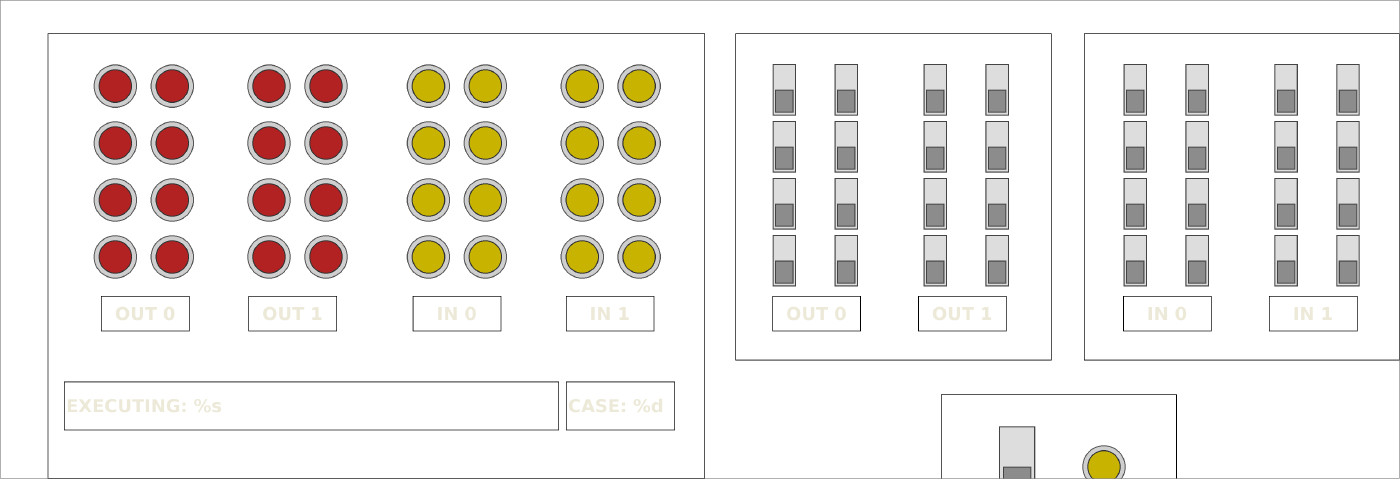
VISUALIZATION StandardPLCversenyVISU  // 1967x673
    Rectangle (1322,554 331x259)
    Rectangle (1033,47 444x459)
    Rectangle (67,47 923x626)
    Lamp1 (127,86 70x70), variable: GIOL.out0, style: Lamp-Lamp1-Red
    Lamp1 (207,86 70x70), variable: GIOL.out1, style: Lamp-Lamp1-Red
    Lamp1 (343,86 70x70), variable: GIOL.out8, style: Lamp-Lamp1-Red
    Lamp1 (423,86 70x70), variable: GIOL.out9, style: Lamp-Lamp1-Red
    Lamp1 (127,166 70x70), variable: GIOL.out2, style: Lamp-Lamp1-Red
    Lamp1 (207,166 70x70), variable: GIOL.out3, style: Lamp-Lamp1-Red
    Lamp1 (343,166 70x70), variable: GIOL.out10, style: Lamp-Lamp1-Red
    Lamp1 (423,166 70x70), variable: GIOL.out11, style: Lamp-Lamp1-Red
    Lamp1 (127,246 70x70), variable: GIOL.out4, style: Lamp-Lamp1-Red
    Lamp1 (207,246 70x70), variable: GIOL.out5, style: Lamp-Lamp1-Red
    Lamp1 (343,246 70x70), variable: GIOL.out12, style: Lamp-Lamp1-Red
    Lamp1 (423,246 70x70), variable: GIOL.out13, style: Lamp-Lamp1-Red
    Lamp1 (127,326 70x70), variable: GIOL.out6, style: Lamp-Lamp1-Red
    Lamp1 (207,326 70x70), variable: GIOL.out7, style: Lamp-Lamp1-Red
    Lamp1 (343,326 70x70), variable: GIOL.out14, style: Lamp-Lamp1-Red
    Lamp1 (423,326 70x70), variable: GIOL.out15, style: Lamp-Lamp1-Red
    Lamp1 (567,86 70x70), variable: GIOL.in0, style: Lamp-Lamp1-Yellow
    Lamp1 (647,86 70x70), variable: GIOL.in1, style: Lamp-Lamp1-Yellow
    Lamp1 (783,86 70x70), variable: GIOL.in8, style: Lamp-Lamp1-Yellow
    Lamp1 (863,86 70x70), variable: GIOL.in9, style: Lamp-Lamp1-Yellow
    Lamp1 (567,166 70x70), variable: GIOL.in2, style: Lamp-Lamp1-Yellow
    Lamp1 (647,166 70x70), variable: GIOL.in3, style: Lamp-Lamp1-Yellow
    Lamp1 (783,166 70x70), variable: GIOL.in10, style: Lamp-Lamp1-Yellow
    Lamp1 (863,166 70x70), variable: GIOL.in11, style: Lamp-Lamp1-Yellow
    Lamp1 (567,246 70x70), variable: GIOL.in4, style: Lamp-Lamp1-Yellow
    Lamp1 (647,246 70x70), variable: GIOL.in5, style: Lamp-Lamp1-Yellow
    Lamp1 (783,246 70x70), variable: GIOL.in12, style: Lamp-Lamp1-Yellow
    Lamp1 (863,246 70x70), variable: GIOL.in13, style: Lamp-Lamp1-Yellow
    Lamp1 (567,326 70x70), variable: GIOL.in6, style: Lamp-Lamp1-Yellow
    Lamp1 (647,326 70x70), variable: GIOL.in7, style: Lamp-Lamp1-Yellow
    Lamp1 (783,326 70x70), variable: GIOL.in14, style: Lamp-Lamp1-Yellow
    Lamp1 (863,326 70x70), variable: GIOL.in15, style: Lamp-Lamp1-Yellow
    Rectangle (349,416 124x49), "OUT 1"
    Rectangle (580,416 124x49), "IN 0"
    Rectangle (142,416 124x49), "OUT 0"
    Rectangle (795,416 124x49), "IN 1"
    Rectangle (90,536 695x68), "EXECUTING: %s", text variable: GIOL.TaskName
    DipSwitch (1153,86 72x80), variable: GIOL.out1, behaviour: TOGGLE, style: Switch-DipSwitch-Gray
    DipSwitch (1066,86 72x80), variable: GIOL.out0, behaviour: TOGGLE, style: Switch-DipSwitch-Gray
    DipSwitch (1153,166 72x80), variable: GIOL.out3, behaviour: TOGGLE, style: Switch-DipSwitch-Gray
    DipSwitch (1066,166 72x80), variable: GIOL.out2, behaviour: TOGGLE, style: Switch-DipSwitch-Gray
    DipSwitch (1153,246 72x80), variable: GIOL.out5, behaviour: TOGGLE, style: Switch-DipSwitch-Gray
    DipSwitch (1066,246 72x80), variable: GIOL.out4, behaviour: TOGGLE, style: Switch-DipSwitch-Gray
    DipSwitch (1153,326 72x80), variable: GIOL.out7, behaviour: TOGGLE, style: Switch-DipSwitch-Gray
    DipSwitch (1066,326 72x80), variable: GIOL.out6, behaviour: TOGGLE, style: Switch-DipSwitch-Gray
    DipSwitch (1365,86 72x80), variable: GIOL.out9, behaviour: TOGGLE, style: Switch-DipSwitch-Gray
    DipSwitch (1278,86 72x80), variable: GIOL.out8, behaviour: TOGGLE, style: Switch-DipSwitch-Gray
    DipSwitch (1365,166 72x80), variable: GIOL.out11, behaviour: TOGGLE, style: Switch-DipSwitch-Gray
    DipSwitch (1278,166 72x80), variable: GIOL.out10, behaviour: TOGGLE, style: Switch-DipSwitch-Gray
    DipSwitch (1365,246 72x80), variable: GIOL.out13, behaviour: TOGGLE, style: Switch-DipSwitch-Gray
    DipSwitch (1278,246 72x80), variable: GIOL.out12, behaviour: TOGGLE, style: Switch-DipSwitch-Gray
    DipSwitch (1365,326 72x80), variable: GIOL.out15, behaviour: TOGGLE, style: Switch-DipSwitch-Gray
    DipSwitch (1278,326 72x80), variable: GIOL.out14, behaviour: TOGGLE, style: Switch-DipSwitch-Gray
    Rectangle (1290,416 124x49), "OUT 1"
    Rectangle (1085,416 124x49), "OUT 0"
    Rectangle (1523,47 444x459)
    DipSwitch (1646,86 72x80), variable: GIOL.bIn1, behaviour: TOGGLE, style: Switch-DipSwitch-Gray
    DipSwitch (1559,86 72x80), variable: GIOL.bIn0, behaviour: TOGGLE, style: Switch-DipSwitch-Gray
    DipSwitch (1646,166 72x80), variable: GIOL.bIn3, behaviour: TOGGLE, style: Switch-DipSwitch-Gray
    DipSwitch (1559,166 72x80), variable: GIOL.bIn2, behaviour: TOGGLE, style: Switch-DipSwitch-Gray
    DipSwitch (1646,246 72x80), variable: GIOL.bIn5, behaviour: TOGGLE, style: Switch-DipSwitch-Gray
    DipSwitch (1559,246 72x80), variable: GIOL.bIn4, behaviour: TOGGLE, style: Switch-DipSwitch-Gray
    DipSwitch (1646,326 72x80), variable: GIOL.bIn7, behaviour: TOGGLE, style: Switch-DipSwitch-Gray
    DipSwitch (1559,326 72x80), variable: GIOL.bIn6, behaviour: TOGGLE, style: Switch-DipSwitch-Gray
    DipSwitch (1858,86 72x80), variable: GIOL.bIn9, behaviour: TOGGLE, style: Switch-DipSwitch-Gray
    DipSwitch (1771,86 72x80), variable: GIOL.bIn8, behaviour: TOGGLE, style: Switch-DipSwitch-Gray
    DipSwitch (1858,166 72x80), variable: GIOL.bIn11, behaviour: TOGGLE, style: Switch-DipSwitch-Gray
    DipSwitch (1771,166 72x80), variable: GIOL.bIn10, behaviour: TOGGLE, style: Switch-DipSwitch-Gray
    DipSwitch (1858,246 72x80), variable: GIOL.bIn13, behaviour: TOGGLE, style: Switch-DipSwitch-Gray
    DipSwitch (1771,246 72x80), variable: GIOL.bIn12, behaviour: TOGGLE, style: Switch-DipSwitch-Gray
    DipSwitch (1858,326 72x80), variable: GIOL.bIn15, behaviour: TOGGLE, style: Switch-DipSwitch-Gray
    DipSwitch (1771,326 72x80), variable: GIOL.bIn14, behaviour: TOGGLE, style: Switch-DipSwitch-Gray
    Rectangle (1783,416 124x49), "IN 1"
    Rectangle (1578,416 124x49), "IN 0"
    Rectangle (795,536 153x68), "CASE: %d", text variable: GIOL.CaseNum
    DipSwitch (1371,599 116x113), variable: MAIN.INMODE.INState, behaviour: TOGGLE, style: Switch-DipSwitch-Gray
    Rectangle (1381,744 226x49), "INPUT MODE"
    Lamp1 (1516,621 70x70), variable: MAIN.INMODE.INState, style: Lamp-Lamp1-Yellow
END_VISUALIZATION

(* stored: Version 1.1.0.1, ProductVersion 3.1.4024.15
   Visu StandardPLCversenyVISU: Id {a8bc012b-8952-461b-92ed-7c0d35e309be} *)
